# B&R Automation Studio project TD52 (part 140)

#### Ctr_OutVRDPCyclic.st
```iecst
(*******************************************************************************
Ctr_OutlVentRDP		controller engine room differential pressure with outlet ventilation fan(s)

This code is confidential and proprietary to the INNIO Company.
It may not be used in any form, or reproduced in any manner,
without the express written permission of the INNIO Company.
Copyright, INNIO Company, 2022

Customized modifications: -
------------------------

History:
-------
V4.04.0		06.10.2016	Stary			created
			02.11.2016	lettenb.		% scaling corr., cleanup
			15.11.2016  Stary		    added manual operation aux-control for outlet-ventilation
			04.01.2017  Stary           correction of task after test on simulator
V4.11.0		28.01.2022	Perktold		included plant controller upgrade

Specification       : PID-controller for outlet ventilation fan(s) to ensure a constant room differential pressure

Instructions for use: Modify release/X/external Y customized when needed
--------------------

Outstandings:
------------
(*******************************************************************************)

PROGRAM _CYCLIC

	(* Parameter *)
	Para.tCtr_OutlVE_RDP.W_set;
	Para.tCtr_OutlVE_RDP.W_set2;
	Para.tCtr_OutlVE_RDP.W_min;
	Para.tCtr_OutlVE_RDP.W_max;
	Para.tCtr_OutlVE_RDP.dW_up;
	Para.tCtr_OutlVE_RDP.dW_down;
	Para.tCtr_OutlVE_RDP.deadband;
	Para.tCtr_OutlVE_RDP.Y_min;
	Para.tCtr_OutlVE_RDP.Y_max;
	Para.tCtr_OutlVE_RDP.dY_max;
	Para.tCtr_OutlVE_RDP.Y_block;
	Para.tCtr_OutlVE_RDP.invert;
	Para.tCtr_OutlVE_RDP.Kp;
	Para.tCtr_OutlVE_RDP.Tn;
	Para.tCtr_OutlVE_RDP.Tv;
	Para.tCtr_OutlVE_RDP.Kp_GainScheduling;
	Para.tCtr_OutlVE_RDP.Tn_GainScheduling;
	Para.tCtr_OutlVE_RDP.Tv_GainScheduling;
	Para.tCtr_OutlVE_RDP.t_min_pulse_down;
	Para.tCtr_OutlVE_RDP.t_min_pulse_up;
	Para.tCtr_OutlVE_RDP.t_period_down;
	Para.tCtr_OutlVE_RDP.t_period_up;

	(* Time delay door-contact, to wait for correct measuring value room differential pressure after MSF --> avoid jump of Y *)
	TON_DC(IN := IN_VE.tER_DoorClosed.Di , PT := T#5s);
	bTON_DoorContact := TON_DC.Q;

	(* Input variables *)
	tCtr_OutlVE_RDP_In	 		:= VIS2MM.tCtr_OutlVE_RDP_In;

	(* Input from module *)
	tCtr_OutlVE_RDP_In.enable	:=	IN_VE.tPB2MM.bParaSetupOk		(* enable controller *)
							AND	    Para.bCtr_OutlVE_RDP
							AND     OUT_VE.tRel_ER_FC.Do
							AND	    RTM25
							AND     OUT_VE.tRel_ER_Fan.Do
							AND		bTON_DoorContact
							AND NOT MM2VIS.bMsg3367
							AND NOT MM2VIS.bMsg2705
							AND NOT bCtrER_YFix;

	tCtr_OutlVE_RDP_In.W_ext_Active		:= FALSE;		(* select external W *) //from visu
	tCtr_OutlVE_RDP_In.W_ext        	:= 0;
	tCtr_OutlVE_RDP_In.W_set2_Active	:= FALSE;		(*Input to define which internal setpoint will be used TRUE = use the 2nd set point | FALSE use the normal "1st" one*)
	tCtr_OutlVE_RDP_In.GainScheduling	:= 0.0;			(*Input for Gain Scheduling: 0.0 = use 100% of the Standard PID-Parameters | 1.0 = use 100% of the GainSched. PID Parameters | linear interpolation in between*)
	tCtr_OutlVE_RDP_In.Y_min_cust		:= -1.0;		(*"customized" Y-Min at the current moment (The existing Y-Min parameter is the global minimum. To have an effect Y_min_cust needs to be > the parameter | -1.0 = function not used*)
	tCtr_OutlVE_RDP_In.Y_max_cust		:= 1.0;			(*"customized" Y-Max at the current moment (The existing Y-Max parameter is the global maximum. To have an effect Y_max_cust needs to be < the parameter | 1.0 = function not used*)
	tCtr_OutlVE_RDP_In.Retrigger		:= FALSE;		(*a rising edge on this input signals the controller to retrigger - set W on X and force the Integrator to the current Y*)
	tCtr_OutlVE_RDP_In.A;								(*optional: feed forward Input*)

	(* Special operation-modes of PID-controller *)

		// Gas-pre-alarm/gas-alarm:
		    (* use of external Yset --> totally open the louver(s) *)
				IF IN_VE.bMsg1052 OR IN_VE.bMsg1053 THEN
					tCtr_OutlVE_RDP_In.Y_set_Active := TRUE;
					tCtr_OutlVE_RDP_In.Y_set := 1.0;
					RAMPE_Y_set_intern := FALSE;

		// Fire-alarm:
			(* use of external Yset --> totally close the louver(s) *)
				ELSIF IN_VE.bMsg1054 THEN
					tCtr_OutlVE_RDP_In.Y_set_Active := TRUE;
					tCtr_OutlVE_RDP_In.Y_set := 0.0;
					RAMPE_Y_set_intern := FALSE;

		// Engine room door-sensors tripped:
			(* use of internal Yset = last setpoint when ctr was active + slow PID-ramp *)
				ELSIF NOT bTON_DoorContact THEN
					tCtr_OutlVE_RDP_In.Y_set_Active := TRUE;
					Y_set_intern := rCtr_OutlVe_RDP_Y_old;  (* guilty for max. 15s, if doors are longer open then shutdown with bMsg3367 *)
					RAMPE_Y_set_intern := TRUE;

		// Measuring signal failure room differential pressure:
			(* use of internal Yset = ctr-signal from inlet ventilation + offset-para [13586] + slow PID-ramp *)
				ELSIF MM2VIS.bMsg2705 THEN
					tCtr_OutlVE_RDP_In.Y_set_Active := TRUE;
					Y_set_intern := tCtr_ER_Out.Y + (Para.rVent_SpeedDif);
					RAMPE_Y_set_intern := TRUE;

		// Manual operating auxiliaries control - Handbedienebene
				ELSIF (NOT tCtr_OutlVE_RDP_In.enable AND OUT_VE.tRel_ER_FC.Do AND IN_VE.tManAuxCtr.bER_OutlV_FC_Set) THEN
					tCtr_OutlVE_RDP_In.Y_set_Active  := TRUE;
					tCtr_OutlVE_RDP_In.Y_set         := IN_VE.tManAuxCtr.rER_OutlV_FC_Set;
					RAMPE_Y_set_intern := FALSE;

		// normal PID mode
				ELSE
					tCtr_OutlVE_RDP_In.Y_set_Active := FALSE;
					RAMPE_Y_set_intern := FALSE;
					Y_set_intern := tCtr_OutlVE_RDP_Out.Y;
				END_IF;

	(* slow PID-ramp *)
		RAMPE_R_0(enable := TRUE, In := Y_set_intern, Rise := 0.01, Sink := 0.01, TC_Time := 100);

		IF RAMPE_Y_set_intern THEN
			tCtr_OutlVE_RDP_In.Y_set := RAMPE_R_0.Out;
		END_IF

	tCtr_OutlVE_RDP_In.X := IN_VE.tPrDiff_ER.Ai;				(* select X *)

	(* add offset to Y *)
	xSigScal_R_CtrRDP_CtrER.X  := tCtr_ER_Out.Y;				(* scaling from setpoint ctr engine room to offset for use in outlet ventilation ctr *)
	xSigScal_R_CtrRDP_CtrER.X1 := Para.rScal_CtrInlVentER_Set_Min;
	xSigScal_R_CtrRDP_CtrER.X2 := Para.rScal_CtrInlVentER_Set_Max;
	xSigScal_R_CtrRDP_CtrER.Y1 := Para.rScal_OffSetMin_CtrOutlVent;
	xSigScal_R_CtrRDP_CtrER.Y2 := Para.rScal_OffSetMax_CtrOutlVent;
	xSigScal_R_CtrRDP_CtrER();

	xSigScal_R_CtrRDP_EngP.X  := IN_VE.rP_Act_Norm_Filt;		(* scaling from actual engine power to offset for use in outlet ventilation ctr *)
	xSigScal_R_CtrRDP_EngP.X1 := Para.rScal_PminEl;
	xSigScal_R_CtrRDP_EngP.X2 := Para.rScal_PmaxEl;
	xSigScal_R_CtrRDP_EngP.Y1 := Para.rScal_OffSetMin_Pel;
	xSigScal_R_CtrRDP_EngP.Y2 := Para.rScal_OffSetMax_Pel;
	xSigScal_R_CtrRDP_EngP();

	(* Input from Visualization via OPC *)
	tCtr_OutlVE_RDP_In.Y_man_Active;
	tCtr_OutlVE_RDP_In.Y_man;
	tCtr_OutlVE_RDP_In.X_min;
	tCtr_OutlVE_RDP_In.X_max;
	tCtr_OutlVE_RDP_In.Tune_quality;
	tCtr_OutlVE_RDP_In.Tune_PI;
	tCtr_OutlVE_RDP_In.Tune_PID;
	tCtr_OutlVE_RDP_In.Tune_start;
	tCtr_OutlVE_RDP_In.Tune_stop;
	tCtr_OutlVE_RDP_In.Tune_takeover;

	xCtr_OutlVE_RDP();

	(* Writing of actual Y on internal variable *)

	IF bTON_DoorContact THEN
		rCtr_OutlVe_RDP_Y_old	        := tCtr_OutlVE_RDP_Out.Y;	(* used as setpoint if engine room door-sensors have tripped *)
	END_IF;

	(* Output variables function block *)
	(* Output to module(s) *)

		// Control of outlet ventilation speed depending on ctr-signal inlet ventilation:
		// --> activation with parameter [13846]
			IF tCtr_OutlVE_RDP_In.enable AND Para.bCtr_RDP_OutlVE_Dep_InlVent AND NOT Para.bCtr_RDP_OutlVE_Dep_EngP THEN
				OUT_VE.tCtr_OutlVE_RDP_Set.Ao := LIMIT(0.0, tCtr_OutlVE_RDP_Out.Y + xSigScal_R_CtrRDP_CtrER.Y_SCAL, 1.0); (* analog out *)

		// Control of outlet ventilation speed depending on actual engine power:
		// --> activation with parameter [13847]
			ELSIF tCtr_OutlVE_RDP_In.enable AND Para.bCtr_RDP_OutlVE_Dep_EngP AND NOT Para.bCtr_RDP_OutlVE_Dep_InlVent THEN
				OUT_VE.tCtr_OutlVE_RDP_Set.Ao := LIMIT(0.0, tCtr_OutlVE_RDP_Out.Y + xSigScal_R_CtrRDP_EngP.Y_SCAL, 1.0); (* analog out *)

		// Control of outlet ventilation speed depending on inlet ventilation and actual engine power:
		// --> activation with parameter [1346+13847]
			ELSIF tCtr_OutlVE_RDP_In.enable AND Para.bCtr_RDP_OutlVE_Dep_InlVent AND Para.bCtr_RDP_OutlVE_Dep_EngP THEN
				OUT_VE.tCtr_OutlVE_RDP_Set.Ao := LIMIT(0.0, tCtr_OutlVE_RDP_Out.Y + xSigScal_R_CtrRDP_CtrER.Y_SCAL + xSigScal_R_CtrRDP_EngP.Y_SCAL, 1.0); (* analog out *)

			ELSE
				OUT_VE.tCtr_OutlVE_RDP_Set.Ao   := tCtr_OutlVE_RDP_Out.Y;		(* analog out *)
			END_IF;

	(* Output to Visualization via OPC *)
	MM2VIS.tCtr_OutlVE_RDP_Out		:= tCtr_OutlVE_RDP_Out;
	MM2VIS.rCtr_OutlVE_RDP_Set      := OUT_VE.tCtr_OutlVE_RDP_Set.Ao;
	VIS2MM.tCtr_OutlVE_RDP_In		:= tCtr_OutlVE_RDP_In;		(* write back to IN_struct for reset: Tune_takeover, X-display, ...!*)

	tCtr_OutlVE_RDP_Out.Active;
	tCtr_OutlVE_RDP_Out.Y;
	tCtr_OutlVE_RDP_Out.W;
	tCtr_OutlVE_RDP_Out.e;
	tCtr_OutlVE_RDP_Out.Kp_tune;
	tCtr_OutlVE_RDP_Out.Tn_tune;
	tCtr_OutlVE_RDP_Out.Tv_tune;
	tCtr_OutlVE_RDP_Out.status;
	tCtr_OutlVE_RDP_Out.Step_down;
	tCtr_OutlVE_RDP_Out.Step_up;

END_PROGRAM
```

#### Ctr_OutVRDPInit.st
```iecst
PROGRAM _INIT

	xCtr_OutlVE_RDP.pParameter 	:= ADR(Para.tCtr_OutlVE_RDP);
	xCtr_OutlVE_RDP.pInput 	 	:= ADR(tCtr_OutlVE_RDP_In);
	xCtr_OutlVE_RDP.pOutput	 	:= ADR(tCtr_OutlVE_RDP_Out);

	tCtr_OutlVE_RDP_In.AlwaysUseYRamp		:= TRUE;	(*If TRUE the Y signal will always limit the change rate via the according parameter | if FALSE the Y signal will jump in case the controller is disabled (blocked or set)*)
	tCtr_OutlVE_RDP_In.KeepYManAtBlock		:= TRUE;	(*If TRUE the controller will keep the Y-man value constant in case the controller is disabled (blocked or set) | If FALSE the blocked or set value will override the Y-man value*)
	tCtr_OutlVE_RDP_In.Y_min_cust			:= -1.0;	(*"customized" Y-Min at the current moment (The existing Y-Min parameter is the global minimum. To have an effect Y_min_cust needs to be > the parameter | -1.0 = function not used*)
	tCtr_OutlVE_RDP_In.Y_max_cust			:=  1.0;	(*"customized" Y-Max at the current moment (The existing Y-Max parameter is the global maximum. To have an effect Y_max_cust needs to be < the parameter | 1.0 = function not used*)
	tCtr_OutlVE_RDP_In.StepperMode			:= FALSE;	(* TRUE = use PWM-Mode (standard mode until 4.10) | FALSE = use continuous servo drive *)

END_PROGRAM
```

#### Ctr_OutVRDP.var
```iecst
VAR
	rCtr_OutlVe_RDP_Y_old : REAL; (*write the actual Y on this internal variable*)
	xSigScal_R_CtrRDP_EngP : xSigScal_R := (0);
	xSigScal_R_CtrRDP_CtrER : xSigScal_R := (0);
	TON_DC : TON; (*TON door contact*)
	RAMPE_R_0 : RAMPE_R := (0);
	RAMPE_Y_set_intern : BOOL := 0;
	Y_set_intern : REAL;
END_VAR
```

### Program Logical/Ventilation/Ctr_ER (IEC, version 4.11.0) - controller engine room temperature

#### Ctr_ERCyclic.st
```iecst
(*******************************************************************************
Ctr_ER		controller engine room temperature

This code is confidential and proprietary to the INNIO Company.
It may not be used in any form, or reproduced in any manner,
without the express written permission of the INNIO Company.
Copyright, INNIO Company, 2022

Customized modifications: -
------------------------

History:
-------
V0.00.0		17.04.2012	lettenbichler	created
			23.11.2012	lettenbichler	write back to IN_struct added (zengerer)
V3.99.0		24.06.2013	lettenbichler	tCtr_ER_In.Y_set := 100.0 -> 1.0, bugfix
V4.00.0		22.05.2015					tCtr_ER_In.X: Para.bT_InAirER_Active added(room vent.to 100% if no sensor active)
V4.03.0 	07.08.2015  Denk			Manual operating auxiliaries control functionality added
V4.05.0 	20.09.2017	Messner			Active Cooling Program added
V4.11.0		28.01.2022	Perktold		included plant controller upgrade

Instructions for use:
--------------------

Outstandings:
------------
(*******************************************************************************)

PROGRAM _CYCLIC

	(* Parameter *)
	Para.tCtr_ER.W_set;
	Para.tCtr_ER.W_set2;
	Para.tCtr_ER.W_min;
	Para.tCtr_ER.W_max;
	Para.tCtr_ER.dW_up;
	Para.tCtr_ER.dW_down;
	Para.tCtr_ER.deadband;
	Para.tCtr_ER.Y_min;
	Para.tCtr_ER.Y_max;
	Para.tCtr_ER.dY_max;
	Para.tCtr_ER.Y_block;
	Para.tCtr_ER.invert;
	Para.tCtr_ER.Kp;
	Para.tCtr_ER.Tn;
	Para.tCtr_ER.Tv;
	Para.tCtr_ER.Kp_GainScheduling;
	Para.tCtr_ER.Tn_GainScheduling;
	Para.tCtr_ER.Tv_GainScheduling;
	Para.tCtr_ER.t_min_pulse_down;
	Para.tCtr_ER.t_min_pulse_up;
	Para.tCtr_ER.t_period_down;
	Para.tCtr_ER.t_period_up;

	(* Input variables *)
	tCtr_ER_In	 				:= VIS2MM.tCtr_ER_In;

	(* Input from module *)
	tCtr_ER_In.enable			:=	IN_VE.tPB2MM.bParaSetupOk		(* enable controller *)
							AND		Para.bCtr_ER
							AND 	OUT_VE.tRel_ER_FC.Do
							AND	  ((RTM25 AND OUT_VE.tRel_ER_Fan.Do) OR (Para.bER_VentColdCountryMode AND NOT OUT_VE.tSet_ER_Fan_Min.Do))
							AND NOT MS_LUE
							AND NOT bCtrER_YFix;

	tCtr_ER_In.W_ext_Active	:= tCtr_ER_In.W_ext_Active OR TRUE;		(* select external W *) //from visu

	IF IN_VE.bEng_Aux_Dem_CDR THEN
		tCtr_ER_In.W_ext :=	 Para.rT_CtrER_WexRun;					(* external W *)
	ELSIF IN_VE.bACP_AirER_Dem THEN
		tCtr_ER_In.W_ext :=	 Para.rT_ACP_AirER_sp;					(* ACP  Room Temperature set point *)
	ELSE
		tCtr_ER_In.W_ext :=	 Para.rT_CtrER_WexStop;
	END_IF;
	tCtr_ER_In.W_set2_Active	:= FALSE;		(*Input to define which internal setpoint will be used TRUE = use the 2nd set point | FALSE use the normal "1st" one*)
	tCtr_ER_In.GainScheduling	:= 0.0;			(*Input for Gain Scheduling: 0.0 = use 100% of the Standard PID-Parameters | 1.0 = use 100% of the GainSched. PID Parameters | linear interpolation in between*)
	tCtr_ER_In.Y_min_cust		:= -1.0;		(*"customized" Y-Min at the current moment (The existing Y-Min parameter is the global minimum. To have an effect Y_min_cust needs to be > the parameter | -1.0 = function not used*)
	tCtr_ER_In.Y_max_cust		:= 1.0;			(*"customized" Y-Max at the current moment (The existing Y-Max parameter is the global maximum. To have an effect Y_max_cust needs to be < the parameter | 1.0 = function not used*)
	tCtr_ER_In.Retrigger		:= FALSE;		(*a rising edge on this input signals the controller to retrigger - set W on X and force the Integrator to the current Y*)
	tCtr_ER_In.A;								(*optional: feed forward Input*)

	IF bCtrER_YFix = TRUE THEN
		tCtr_ER_In.Y_set_Active	:= bCtrER_YFix; 	 				(* select external Y *)
		tCtr_ER_In.Y_set		:= 1.0;
	ELSIF (	NOT tCtr_ER_In.enable 									(* Manual operating auxiliaries control - Handbedienebene *)
			AND OUT_VE.tRel_ER_FC.Do
			AND IN_VE.tManAuxCtr.bER_FC_Set) THEN
		tCtr_ER_In.Y_set_Active := TRUE;
		tCtr_ER_In.Y_set		:= IN_VE.tManAuxCtr.rER_FC_Set;
	ELSE
		tCtr_ER_In.Y_set_Active	:= FALSE;
	END_IF;

	IF Para.bER_VentColdCountryMode AND IN_VE.bEng_Aux_Dem_CDR (*AND Para.bT_InAirER_Active*) THEN
		tCtr_ER_In.X :=	MAX(rT_AirER, IN_VE.rT_Ch_T1LP_Avg);		(* select X *)
	ELSE
		tCtr_ER_In.X :=	    rT_AirER;
	END_IF;
	tCtr_ER_In.A := 0;

	(* Input from Visualization via OPC *)
	tCtr_ER_In.Y_man_Active;
	tCtr_ER_In.Y_man;
	tCtr_ER_In.X_min;
	tCtr_ER_In.X_max;
	tCtr_ER_In.Tune_quality;
	tCtr_ER_In.Tune_PI;
	tCtr_ER_In.Tune_PID;
	tCtr_ER_In.Tune_start;
	tCtr_ER_In.Tune_stop;
	tCtr_ER_In.Tune_takeover;

	xCtr_ER();

	(* Output variables function block *)
	(* Output to module(s) *)
	OUT_VE.tER_FC_Set.Ao 	:= tCtr_ER_Out.Y;	(* analog out *)

	(* Output to Visualization via OPC *)
	MM2VIS.tCtr_ER_Out		:= tCtr_ER_Out;
	VIS2MM.tCtr_ER_In		:= tCtr_ER_In;		(* write back to IN_struct for reset: Tune_takeover, X-display, ...!*)

	tCtr_ER_Out.Active;
	tCtr_ER_Out.Y;
	tCtr_ER_Out.W;
	tCtr_ER_Out.e;
	tCtr_ER_Out.Kp_tune;
	tCtr_ER_Out.Tn_tune;
	tCtr_ER_Out.Tv_tune;
	tCtr_ER_Out.status;
	tCtr_ER_Out.Step_down;
	tCtr_ER_Out.Step_up;

END_PROGRAM
```

#### Ctr_ERInit.st
```iecst
PROGRAM _INIT

	xCtr_ER.pParameter 	:= ADR(Para.tCtr_ER);
	xCtr_ER.pInput 	 	:= ADR(tCtr_ER_In);
	xCtr_ER.pOutput	 	:= ADR(tCtr_ER_Out);

	tCtr_ER_In.AlwaysUseYRamp		:= TRUE;	(*If TRUE the Y signal will always limit the change rate via the according parameter | if FALSE the Y signal will jump in case the controller is disabled (blocked or set)*)
	tCtr_ER_In.KeepYManAtBlock		:= TRUE;	(*If TRUE the controller will keep the Y-man value constant in case the controller is disabled (blocked or set) | If FALSE the blocked or set value will override the Y-man value*)
	tCtr_ER_In.Y_min_cust			:= -1.0;	(*"customized" Y-Min at the current moment (The existing Y-Min parameter is the global minimum. To have an effect Y_min_cust needs to be > the parameter | -1.0 = function not used*)
	tCtr_ER_In.Y_max_cust			:=  1.0;	(*"customized" Y-Max at the current moment (The existing Y-Max parameter is the global maximum. To have an effect Y_max_cust needs to be < the parameter | 1.0 = function not used*)
	tCtr_ER_In.StepperMode			:= FALSE;	(* TRUE = use PWM-Mode (standard mode until 4.10) | FALSE = use continuous servo drive *)

END_PROGRAM
```

### Program Logical/Ventilation/vis_VE (IEC, version 4.05.1) - visualization

#### vis_VECyclic.st
```iecst
(*******************************************************************************
vis			visualization

This code is confidential and proprietary to the INNIO Company.
It may not be used in any form, or reproduced in any manner,
without the express written permission of the INNIO Company.
Copyright, INNIO Company, 2019

Customized modifications: -
------------------------

History:
-------
V3.99.0	24.04.2012	lettenb.	new
V4.00.0	02.06.2014				MM2VIS.bRel_ER_Fan: OUT_VE.tRel_ER_Fan.Do -> OUT_VE.tRel_ER_FC.Do, bugfix
V4.03.0 19.11.2015  Stary       added MM2VIS.rPrDiff_ER :=  IN_VE.tPrDiff_ER.Ai;
V4.04.0 21.10.2016  Stary       added MM2VIS.bCtrER_YFix :=  bCtrER_YFix; for visualization of BOP on HMI
V4.04.0 22.10.2016  Stary       added status-messages of fire-protection flaps
		07.11.2016	lettenb.	MM2VIS.rP_Red_T_InAirER_Norm removed(see:OpState)
V4.04.0 09.01.2017  Stary       correction of line 43 (was written on status of fire prot flap outlet air 1 too)
V4.05.1 01.03.2018	lettenb.	Pos_InlLou1_OK, Pos_InlLou2_OK, Pos_OutlLou1_OK added(kluckner), bugfix

Instructions for use:
--------------------
Outstandings:
------------
*******************************************************************************)
PROGRAM _CYCLIC

	MM2VIS.rT_AirER							:=	rT_AirER;
	MM2VIS.rPrDiff_ER           			:=  IN_VE.tPrDiff_ER.Ai;

	MM2VIS.bInAirER_Lou1Opened				:=	IN_VE.tInAirER_Lou1Opened.Di OR Pos_InlLou1_OK;
	MM2VIS.bInAirER_Lou2Opened				:=	IN_VE.tInAirER_Lou2Opened.Di OR Pos_InlLou2_OK;
	MM2VIS.bOutAirER_LouOpened				:=	IN_VE.tOutAirER_LouOpened.Di OR Pos_OutlLou1_OK OR Pos_OutlLou2_OK;
	MM2VIS.bInAirER_Fan1DemOn				:=	OUT_VE.tInAirER_Fan1DemOn.Do;
	MM2VIS.bInAirER_Fan2DemOn				:=	OUT_VE.tInAirER_Fan2DemOn.Do;
	MM2VIS.bInAirER_FanSet100				:=	IN_VE.bInAirER_FanSet100;
	MM2VIS.bRel_ER_Fan						:=	OUT_VE.tRel_ER_FC.Do;
	MM2VIS.bCtrER_YFix						:=  bCtrER_YFix;
	MM2VIS.bFireProtFlap1_InlAir_Opened 	:=  IN_VE.tFireProtFlap1_InlAir_Opened.Di AND NOT IN_VE.tFireProtFlap1_InlAir_Closed.Di;
	MM2VIS.bFireProtFlap2_InlAir_Opened 	:=  IN_VE.tFireProtFlap2_InlAir_Opened.Di AND NOT IN_VE.tFireProtFlap2_InlAir_Closed.Di;
	MM2VIS.bFireProtFlap1_OutlAir_Opened 	:=  IN_VE.tFireProtFlap1_OutlAir_Opened.Di AND NOT IN_VE.tFireProtFlap1_OutlAir_Closed.Di;
	MM2VIS.bFireProtFlap2_OutlAir_Opened 	:=  IN_VE.tFireProtFlap2_OutlAir_Opened.Di AND NOT IN_VE.tFireProtFlap2_OutlAir_Closed.Di;

END_PROGRAM
```

### Program Logical/Ventilation/MsgVE (IEC, version 4.13.0) - messages

#### MsgVECyclic.st
```iecst
(*******************************************************************************
MsgVE	 			ventilation messages

This code is confidential and proprietary to the INNIO Company.
It may not be used in any form, or reproduced in any manner,
without written permission of the INNIO Company.
Copyright, INNIO Company, 2022

Customized modifications: -
------------------------

History:
-------
V0.01.0	02.11.2011	lettenb.	new
		18.09.2012	lettenb.	rT_AirER_Customized added (request zengerer)
V3.40.0	17.12.2012	lettenb.	1138 DI_ERV_Op added, preparation for air flow sensor, ATEX
								3224 .PTON := T#0s -> 2s; (W3223 MS & W3224 comes at the same time) bugfix
V3.99.0	19.02.2013	lettenb.	update
		24.05.2013				reset OUT_xx.txx2AB.bGnlTripx changed
V4.00.0	31.01.2014				3367 added, eng.room vent.monit.V3.50
V4.00.1	14.05.2014	lettenb.	1138 var 3/4: FG_FU, ZLVST1 added (MRL kalte laender)
		12.06.2014				3224 xTON_GCB_On.PT:= T#30s -> 300s, bugfix
V4.00.2	16.02.2015				3152,3223 enable with IN_VE.tPB2MM.bSys_Run
V4.03.0 03.08.2015  Stary       added new alarms 2701-2709 FOR controlled louvers
					lettenb.	xMsg2704.Enable: Para.bInlVent_Ctr_OutlLou_Active -> Para.bOutlVent_Ctr_OutlLou_Active, bugfix
		30.09.2015  Stary       2120 tAuxV_Aux_ok added
		23.12.2015	lettenb.	1138 M_DREHZ -> (IN_VE.bEng_Dem OR IN_VE.tEng_Run.Do) to avoid msg after mains failure(restart ability)
V4.04.0 07.07.2016	lettenb.	2630 added(substitution for 1176 in wrong module(CH) tDPr_InAirFilt_Hi -> tDPr_InAirFiltERV_Hi), bugfix
V4.04.0 27.09.2016  Stary       splitted up existing summarized alarms 1138+2120 for ventilation and added single alarms for inlet/outlet --> new messages 2295,2296,2795-2798
		02.11.2016	Tinello		3223 und 3224 deleted --> moved to modul CH
V4.04.0 25.01.2017  Stary   	bugfix after pilot-engines:
								Enable of bMsg2701-bMsg2704 --> deleted Para.bInlVent_Ctr_InlLou_Active cause measuring singnal failure now indepedend OF ventilation type
		01.02.2017	lettenb.	xTON_MonAuxV double function call removed
V4.05.0 30.06.2017	lettenb.	bAuxRel_Louvers added acc. faststart option
		21.12.2017	lettenb.	1138, 2295, 2296 enable alarms depending on existing Di's (stary), bugfix
		22.12.2017	lettenb.	comment added: Safety-related application software source code (EN 13849-1 / 4.6.3)
		22.01.2018	lettenb.	1138 Pos_InlLou1_OK, Pos_InlLou2_OK, Pos_OutlLou1_OK, Pos_OutlLou2_OK added, bugfix
		22.01.2018	lettenb.	3152 bParaSetupOk added TO avoid message at plc startup
		30.01.2018	lettenb.	2706,2707 time delay 10s(fahringer/stary)
V4.06.0	16.07.2018	Perktold,	2968 and 2969 Air inlet/outlet louver status signal failure added
V4.07.0 25.02.2019	Stary/lett. 1138,2295,2296 bAuxRel_FireProtFlaps: FireProtFlap feedback signals included in aux.release, safety case
								2295,2296 bAuxRel_Louvers_... added(same as 1138), xTON_MonAuxV double function call removed, bugfix
V4.10.0 25.01.2021	lettenb.	engine room ventilation not ready - block engine start as long as failure is active, added from task Vent_ER (request fahringer), bugfix
								2120,2795,2796 safety code remark added (request fahringer)
V4.12.0 07.12.2022	lettenb.	2706: IN_VE.tEng_Run.Do added, aggreko -> jenb.standard, #954
V4.13.0 18.03.2024	Bacci		2295: trip used when inlet louvers demanded but not responding (90s)
V4.14.0 10.12.2024	Nagy		New warning 2472 High Temperature Warning and Alarm 9401 Louvers 2024-226

Instructions for use:
--------------------
1) declare alarm with function block "Alm"
	declare buffert alarm bit bMsg<message number>

2) use template to create a new alarm,
   substitue 0000 by alarm number and make settings:

	xMsg0000.Enable		:=	TRUE;		enable/disable alarm
	xMsg0000.Set		:=	FALSE;		alarm set condition
	xMsg0000.PT			:=	T#0s;		alarm delay time
	xMsg0000.Prio		:=	1;			alarm priority: 1-3 = trip, 4 = warning
	xMsg0000.RiskClass	:=	3;			risk class for remote alarm reset acc.TI 1100-0111
	xMsg0000.Reset		:=	FALSE;		FALSE: for all standard alarms	prio 1,2,3 and warnings prio 4
										TRUE : for autoreset alarms

	bMsg0000			:=	xMsg0000.Q;	connect buffert alarm bit for VIS and control

3)  expand INIT

Outstandings:
------------
change bGnlTrip_VE --> bGnlTrip
(*******************************************************************************)
PROGRAM _CYCLIC

	(* reset general trip *)
	OUT_VE.tVE2AB.bGnlTrip1		:=	FALSE;
	OUT_VE.tVE2AB.bGnlTrip2		:=	FALSE;
	OUT_VE.tVE2AB.bGnlTrip3		:=	FALSE;
	OUT_VE.tVE2AB.bGnlWarning	:=	FALSE;
	OUT_VE.tVE2AB.bTriptype1	:=	FALSE;
	OUT_VE.tVE2AB.bTriptype2	:=	FALSE;
	OUT_VE.tVE2AB.bTriptype3	:=	FALSE;

	(*  1135 engine room temperature high *)
	xTON_RoomTemp.IN :=   ((NOT MM2VIS.bMsg3152) AND bT_AirER_Hi)
						OR (NOT Para.bVISA  AND NOT IN_VE.tT_AirER_Ext_Hi.Di);
	xTON_RoomTemp.PT :=  T#30s;
	xTON_RoomTemp();
	T_RTM := xTON_RoomTemp.Q;

	xMsg1135.Enable		:=	TRUE;
	xMsg1135.Set		:= (T_RTM      AND(NOT IN_VE.bEng_Dem_EPS OR IN_VE.bOnly_Island))
						OR (Para.bVISA AND NOT IN_VE.tT_AirER_Ext_Hi.Di);
	xMsg1135.PT			:=	T#0s;

	RTM_VISA := NOT IN_VE.tT_AirER_Ext_Hi.Di  OR (RTM_VISA AND xMsg1135.Q);
	IF Para.bVISA AND RTM_VISA THEN
		xMsg1135.Prio	:=	2;
	ELSE
		xMsg1135.Prio	:=	3;
	END_IF;
	xMsg1135.RiskClass	:=	0;		(* TI 1100-0111 *)
	xMsg1135.Reset		:=	FALSE;
	xMsg1135();
	MM2VIS.bMsg1135	    :=	xMsg1135.Q;

	(*  2472 engine room temperature high warning*)
	xMsg2472.Enable		:=	TRUE;
	xMsg2472.Set		:= bT_AirER_Hi_Wr AND (NOT IN_VE.bEng_Dem_EPS OR IN_VE.bOnly_Island)
	OR (Para.bVISA AND NOT IN_VE.tT_AirER_Ext_Hi.Di);
	xMsg2472.PT			:=	T#1s;
	xMsg2472.Prio		:=	4;
	xMsg2472.RiskClass	:=	0;		(* TI 1100-0111 *)
	xMsg2472.Reset		:=	FALSE;
	xMsg2472();
	MM2VIS.bMsg2472	    :=	xMsg2472.Q;

	(********************************************************************************************************************
	Safety-related application software source code (EN 13849-1 / 4.6.3): BEGIN
	*********************************************************************************************************************)
	(*  1138 engine room fan failure trip (W2120) *)
	bERV_AirFlowMon_Off :=	(IN_VE.tInAirER_Lou1Opened.Di OR IN_VE.tInAirER_Lou2Opened.Di OR IN_VE.tOutAirER_LouOpened.Di OR Pos_InlLou1_OK OR Pos_InlLou2_OK OR Pos_OutlLou1_OK OR Pos_OutlLou2_OK)
					 AND NOT(IN_VE.bEng_Dem OR IN_VE.tEng_Run.Do); 		(* monit.off for reason of natural air flow with open louvers *)
	xTON_StartERV(IN:= IN_VE.bEng_Aux_Dem_CDR, PT:= T#30s);				(* startverzoegerung fuer ueberwachung *)

	IF    Para.bERV_AirFlowMon_Active AND Para.bInAirER_Fan_FU THEN
			(* var: flow sensor, stationaeranlage, container BR6	*)
			(* var: stationaeranlage, steuerung RL durch GEJ inkl. Rueckmeldung RL in Betrieb (flow switch od.IFL 56.32) *)
		xTON_ERV_On(IN:=      FG_FU                        AND NOT IN_VE.tERV_Op.Di AND NOT bERV_AirFlowMon_Off, PT:= T#15s);(* delay on:  eng.room vent.ok/air flow monitoring *)
		xTON_ERV_Of(IN:=  NOT FG_FU                        AND     IN_VE.tERV_Op.Di AND NOT bERV_AirFlowMon_Off, PT:= T#5m); (* delay off: change contact check *)
	ELSIF Para.bERV_AirFlowMon_Active AND NOT Para.bInAirER_Fan_FU THEN
		xTON_ERV_On(IN:=      OUT_VE.tInAirER_Fan1DemOn.Do AND NOT IN_VE.tERV_Op.Di AND NOT bERV_AirFlowMon_Off, PT:= T#15s);(* delay on:  eng.room vent.ok/air flow monitoring *)
		xTON_ERV_Of(IN:=  NOT OUT_VE.tInAirER_Fan1DemOn.Do AND     IN_VE.tERV_Op.Di AND NOT bERV_AirFlowMon_Off, PT:= T#5m); (* delay off: change contact check *)
	ELSIF Para.bInAirER_Fan_FU THEN
			(* var: FU=RUN, ohne luftstromwaechter *)
		xTON_ERV_On(IN:=      FG_FU   					   AND NOT IN_VE.tERV_Op.Di AND    (IN_VE.bEng_Dem OR IN_VE.tEng_Run.Do), PT:= T#15s);
		xTON_ERV_Of(IN:= FALSE, PT:= T#5m);
	ELSE	(* var: lueftung in betrieb, ohne FU, ohne luftstromwaechter *)
		xTON_ERV_On(IN:=      OUT_VE.tInAirER_Fan1DemOn.Do AND NOT IN_VE.tERV_Op.Di AND    (IN_VE.bEng_Dem OR IN_VE.tEng_Run.Do), PT:= T#15s);
		xTON_ERV_Of(IN:= FALSE, PT:= T#5m);
	END_IF;
			(* keine ERV: 	para bERV_AirFlowMon_Active (default =0) => OFF
							para bAirInVentF (default=1) n.r.,
							DI_ERV_Op (default = 1) nicht belegt *)

	bAuxRel_Louvers := (IN_VE.tOutAirER_LouOpened.Di AND IN_VE.tInAirER_Lou1Opened.Di)
					OR((Pos_InlLou1_OK OR Pos_InlLou2_OK) AND (Pos_OutlLou1_OK OR Pos_OutlLou2_OK));

	bAuxRel_FireProtFlaps := IN_VE.tFireProtFlap1_InlAir_Opened.Di  AND IN_VE.tFireProtFlap2_InlAir_Opened.Di AND
							 IN_VE.tFireProtFlap1_OutlAir_Opened.Di AND IN_VE.tFireProtFlap2_OutlAir_Opened.Di;

	xTOF_EngDemEPS(IN:= IN_VE.bEng_Dem_EPS AND NOT IN_VE.tGCB_On.Di, PT:= T#60s);
	bNoMon4BlackStart := xTOF_EngDemEPS.Q AND IN_VE.bEng_Dem_EPS; //T14

	xMsg1138.Enable		:=	IN_VE.tERV_Op.GoodQual;
	xMsg1138.Set		:= (NOT bNoMon4BlackStart AND  ((xTON_ERV_On.Q AND xTON_StartERV.Q)
                                                     OR  xTON_ERV_Of.Q))
						OR (IN_VE.bFS_Act AND xTON_StartERV.Q AND NOT bAuxRel_Louvers)
						OR (IN_VE.bFS_Act AND xTON_StartERV.Q AND NOT bAuxRel_FireProtFlaps);
	xMsg1138.PT			:=	T#0s;
	xMsg1138.Prio		:=	3;
	xMsg1138.RiskClass	:=	4;
	xMsg1138.Reset		:=	FALSE;
	xMsg1138();
	MM2VIS.bMsg1138 	:=	xMsg1138.Q;
	(********************************************************************************************************************
	Safety-related application software source code (EN 13849-1 / 4.6.3): END
	*********************************************************************************************************************)

	(********************************************************************************************************************
	Safety-related application software source code (EN 13849-1 / 4.6.3): BEGIN
	*********************************************************************************************************************)
	(*  2120 engine room fan failure *)
	xTON_MonAuxV(IN:= IN_VE.tGCB_On.Di, PT:= T#60s);		(* release monitoring engine room fan failure *)

	IF Para.bInAirER_Fan_FU THEN
		xTON_ERV.IN			:= (NOT IN_VE.tER_Ext_Err.Di AND     IN_VE.tAuxV_Supply_Ok.Di AND IN_VE.tAuxV_Aux_ok.Di)
							OR (    xTON_MonAuxV.Q	     AND(NOT IN_VE.tAuxV_Supply_Ok.Di
														  OR NOT IN_VE.tAuxV_Aux_ok.Di));
	ELSE
		xTON_ERV.IN			:=  NOT IN_VE.tER_Ext_Err.Di;
	END_IF;
	xTON_ERV(PT:= T#12s);

	xMsg2120.Enable		:=	TRUE;
	xMsg2120.Set		:=	xTON_ERV.Q;
	xMsg2120.PT			:=	T#0s;
	xMsg2120.Prio		:=	4;
	xMsg2120.RiskClass	:=	4;
	xMsg2120.Reset		:=	FALSE;
	xMsg2120();
	MM2VIS.bMsg2120     :=	xMsg2120.Q;

	(* engine room ventilation not ready - block engine start as long as failure is active *)
	OUT_VE.bERV_NotRdy := xMsg2120.Set OR xMsg2795.Set OR xMsg2796.Set;
	(********************************************************************************************************************
	Safety-related application software source code (EN 13849-1 / 4.6.3): END
	*********************************************************************************************************************)

	(********************************************************************************************************************
	Safety-related application software source code (EN 13849-1 / 4.6.3): BEGIN
	*********************************************************************************************************************)
	(*  2295 engine room ventilation failure inlet air *)
	bERV_InlAirFlowMon_Off := (IN_VE.tInAirER_Lou1Opened.Di OR IN_VE.tInAirER_Lou2Opened.Di OR Pos_InlLou1_OK OR Pos_InlLou2_OK)
					  AND NOT (IN_VE.bEng_Dem OR IN_VE.tEng_Run.Do); 	(* monit.off for reason of natural air flow with open louvers *)
	xTON_StartERV(IN:= IN_VE.bEng_Aux_Dem_CDR, PT:= T#30s);				(* startverzoegerung fuer ueberwachung *)

	IF    Para.bERV_AirFlowMon_Active AND Para.bInAirER_Fan_FU THEN
		(* var: flow sensor, stationaeranlage, container BR6	*)
		(* var: stationaeranlage, steuerung RL durch GEJ inkl. Rueckmeldung RL in Betrieb *)
		xTON_ERV_Inl_On(IN:=      FG_FU                        AND NOT IN_VE.tERV_InlAir_Op.Di AND NOT bERV_InlAirFlowMon_Off, PT:= T#15s);(* delay on:  eng.room inl.vent.ok/air flow monitoring *)
		xTON_ERV_Inl_Of(IN:=  NOT FG_FU                        AND     IN_VE.tERV_InlAir_Op.Di AND NOT bERV_InlAirFlowMon_Off, PT:= T#5m); (* delay off: change contact check *)
	ELSIF Para.bERV_AirFlowMon_Active AND NOT Para.bInAirER_Fan_FU THEN
		xTON_ERV_Inl_On(IN:=      OUT_VE.tInAirER_Fan1DemOn.Do AND NOT IN_VE.tERV_InlAir_Op.Di AND NOT bERV_InlAirFlowMon_Off, PT:= T#15s);(* delay on:  eng.room inl.vent.ok/air flow monitoring *)
		xTON_ERV_Inl_Of(IN:=  NOT OUT_VE.tInAirER_Fan1DemOn.Do AND     IN_VE.tERV_InlAir_Op.Di AND NOT bERV_InlAirFlowMon_Off, PT:= T#5m); (* delay off: change contact check *)
	ELSIF Para.bInAirER_Fan_FU THEN
		(* var: FU=RUN, ohne luftstromwaechter *)
		xTON_ERV_Inl_On(IN:=      FG_FU   					   AND NOT IN_VE.tERV_InlAir_Op.Di AND    (IN_VE.bEng_Dem OR IN_VE.tEng_Run.Do), PT:= T#15s);
		xTON_ERV_Inl_Of(IN:= FALSE, PT:= T#5m);
	ELSE	(* var: lueftung in betrieb, ohne FU, ohne luftstromwaechter *)
		xTON_ERV_Inl_On(IN:=      OUT_VE.tInAirER_Fan1DemOn.Do AND NOT IN_VE.tERV_InlAir_Op.Di AND    (IN_VE.bEng_Dem OR IN_VE.tEng_Run.Do), PT:= T#15s);
		xTON_ERV_Inl_Of(IN:= FALSE, PT:= T#5m);
	END_IF;

	bAuxRel_Louvers_InlAir       := IN_VE.tInAirER_Lou1Opened.Di OR Pos_InlLou1_OK OR Pos_InlLou2_OK;
	bAuxRel_FireProtFlaps_InlAir := IN_VE.tFireProtFlap1_InlAir_Opened.Di AND IN_VE.tFireProtFlap2_InlAir_Opened.Di;

	xTOF_EngDemEPS(IN:= IN_VE.bEng_Dem_EPS AND NOT IN_VE.tGCB_On.Di, PT:= T#60s);
	bNoMon4BlackStart := xTOF_EngDemEPS.Q AND IN_VE.bEng_Dem_EPS; //T14

	xTON_InAirER_LouFail(IN:= (OUT_VE.tInAirER_Lou1DemOpen.Do OR OUT_VE.tInAirER_Lou2DemOpen.Do OR OUT_VE.tCtr_InlLou_Set.Ao > 0.5) AND NOT OUT_VE.bInLouRelVE AND xOpMode.Stop,  PT:= T#90s);		(* Inlet louver required and not opened *)

	xMsg2295.Enable		:=	IN_VE.tERV_InlAir_Op.GoodQual OR (xOpMode.Stop AND (xTON_InAirER_LouFail.Q OR MM2VIS.bMsg2295));
	xMsg2295.Set		:=	(NOT bNoMon4BlackStart AND ((xTON_ERV_Inl_On.Q AND xTON_StartERV.Q)
						    OR  xTON_ERV_Inl_Of.Q))
					        OR (IN_VE.bFS_Act AND xTON_StartERV.Q AND NOT bAuxRel_Louvers_InlAir)
	                        OR (IN_VE.bFS_Act AND xTON_StartERV.Q AND NOT bAuxRel_FireProtFlaps_InlAir)
							OR xTON_InAirER_LouFail.Q;
	xMsg2295.PT			:=	T#0s;
	xMsg2295.Prio		:=	3;
	xMsg2295.RiskClass	:=	10;
	xMsg2295.Reset		:=	FALSE;
	xMsg2295();
	MM2VIS.bMsg2295	    :=	xMsg2295.Q;
	OUT_VE.bMsg2295	    :=	xMsg2295.Q;

	(*  2296 engine room ventilation failure outlet air *)
	bERV_OutlAirFlowMon_Off := (IN_VE.tOutAirER_LouOpened.Di OR Pos_OutlLou1_OK OR Pos_OutlLou2_OK)
					   AND NOT (IN_VE.bEng_Dem OR IN_VE.tEng_Run.Do); (* monit.off for reason of natural air flow with open louvers *)
	xTON_StartERV(IN:= IN_VE.bEng_Aux_Dem_CDR, PT:= T#30s);				(* startverzoegerung fuer ueberwachung *)

	IF    Para.bERV_AirFlowMon_Active AND Para.bOutAirER_Fan_FU THEN
		(* var: flow sensor, stationaeranlage, container BR6	*)
		(* var: stationaeranlage, steuerung RL durch GEJ inkl. Rueckmeldung RL in Betrieb *)
		xTON_ERV_Outl_On(IN:=      FG_FU                          AND NOT IN_VE.tERV_OutlAir_Op.Di AND NOT bERV_OutlAirFlowMon_Off, PT:= T#15s);(* delay on:  eng.room outl.vent.ok/air flow monitoring *)
		xTON_ERV_Outl_Of(IN:=  NOT FG_FU                          AND     IN_VE.tERV_OutlAir_Op.Di AND NOT bERV_OutlAirFlowMon_Off, PT:= T#5m); (* delay off: change contact check *)
	ELSIF Para.bERV_AirFlowMon_Active AND NOT Para.bOutAirER_Fan_FU THEN
		xTON_ERV_Outl_On(IN:=      OUT_VE.tOutAirER_LouDemOpen.Do AND NOT IN_VE.tERV_OutlAir_Op.Di AND NOT bERV_OutlAirFlowMon_Off, PT:= T#15s);(* delay on:  eng.room outl.vent.ok/air flow monitoring *)
		xTON_ERV_Outl_Of(IN:=  NOT OUT_VE.tOutAirER_LouDemOpen.Do AND     IN_VE.tERV_OutlAir_Op.Di AND NOT bERV_OutlAirFlowMon_Off, PT:= T#5m); (* delay off: change contact check *)
	ELSIF Para.bOutAirER_Fan_FU THEN
		(* var: FU=RUN, ohne luftstromwaechter *)
		xTON_ERV_Outl_On(IN:=      FG_FU   					      AND NOT IN_VE.tERV_OutlAir_Op.Di AND    (IN_VE.bEng_Dem OR IN_VE.tEng_Run.Do), PT:= T#15s);
		xTON_ERV_Outl_Of(IN:= FALSE, PT:= T#5m);
	ELSE	(* var: lueftung in betrieb, ohne FU, ohne luftstromwaechter *)
		xTON_ERV_Outl_On(IN:=      OUT_VE.tInAirER_Fan1DemOn.Do AND NOT IN_VE.tERV_OutlAir_Op.Di AND    (IN_VE.bEng_Dem OR IN_VE.tEng_Run.Do), PT:= T#15s);
		xTON_ERV_Outl_Of(IN:= FALSE, PT:= T#5m);
	END_IF;

	bAuxRel_Louvers_OutlAir       := IN_VE.tOutAirER_LouOpened.Di OR Pos_OutlLou1_OK OR Pos_OutlLou2_OK;
	bAuxRel_FireProtFlaps_OutlAir := IN_VE.tFireProtFlap1_OutlAir_Opened.Di AND IN_VE.tFireProtFlap2_OutlAir_Opened.Di;

	xTOF_EngDemEPS(IN:= IN_VE.bEng_Dem_EPS AND NOT IN_VE.tGCB_On.Di, PT:= T#60s);
	bNoMon4BlackStart := xTOF_EngDemEPS.Q AND IN_VE.bEng_Dem_EPS; //T14

	xMsg2296.Enable		:=	IN_VE.tERV_OutlAir_Op.GoodQual;
	xMsg2296.Set		:=	(NOT bNoMon4BlackStart AND ((xTON_ERV_Outl_On.Q AND xTON_StartERV.Q)
							OR  xTON_ERV_Outl_Of.Q))
							OR (IN_VE.bFS_Act AND xTON_StartERV.Q AND NOT bAuxRel_Louvers_OutlAir)
							OR (IN_VE.bFS_Act AND xTON_StartERV.Q AND NOT bAuxRel_FireProtFlaps_OutlAir);
	xMsg2296.PT			:=	T#0s;
	xMsg2296.Prio		:=	3;
	xMsg2296.RiskClass	:=	10;
	xMsg2296.Reset		:=	FALSE;
	xMsg2296();
	MM2VIS.bMsg2296	    :=	xMsg2296.Q;
	(********************************************************************************************************************
	Safety-related application software source code (EN 13849-1 / 4.6.3): END
	*********************************************************************************************************************)

	(*  2630 Air inlet filter difference pressure maximum - engine room ventilation *)
	xMsg2630.Enable	   	:= TRUE;
	xMsg2630.Set       	:= NOT IN_VE.tDPr_InAirFiltERV_Hi.Di;
	xMsg2630.PT		   	:= T#0s;
	xMsg2630.Prio	   	:= 4;
	xMsg2630.RiskClass 	:= 4;
	xMsg2630.Reset	   	:= FALSE;
	xMsg2630();
	MM2VIS.bMsg2630		:= xMsg2630.Q;

	(*  2701 measuring signal failure position air inlet louver 1  *)
	xMsg2701.Enable     := IN_VE.tPB2MM.bSys_Run AND Para.bPos_InlLou1_Active;
	xMsg2701.Set        := IN_VE.tPB2MM.bParaSetupOk AND NOT IN_VE.tPos_InlLou1.GoodQual;
	xMsg2701.PT			:=	T#0s;
	xMsg2701.Prio		:=	4;
	xMsg2701.RiskClass	:=	4;
	xMsg2701.Reset		:=	FALSE;
	xMsg2701();
	MM2VIS.bMsg2701		:=	xMsg2701.Q;
	OUT_VE.bMsg2701		:=	xMsg2701.Q;

	(*  2702 measuring signal failure position air inlet louver 2  *)
	xMsg2702.Enable     := IN_VE.tPB2MM.bSys_Run AND Para.bPos_InlLou2_Active;
	xMsg2702.Set        := IN_VE.tPB2MM.bParaSetupOk AND NOT IN_VE.tPos_InlLou2.GoodQual;
	xMsg2702.PT			:=	T#0s;
	xMsg2702.Prio		:=	4;
	xMsg2702.RiskClass	:=	4;
	xMsg2702.Reset		:=	FALSE;
	xMsg2702();
	MM2VIS.bMsg2702		:=	xMsg2702.Q;
	OUT_VE.bMsg2702		:=	xMsg2702.Q;

	(*  2703 measuring signal failure position air outlet louver 1  *)
	xMsg2703.Enable     := IN_VE.tPB2MM.bSys_Run AND Para.bPos_OutlLou1_Active;
	xMsg2703.Set        := IN_VE.tPB2MM.bParaSetupOk AND NOT IN_VE.tPos_OutlLou1.GoodQual;
	xMsg2703.PT			:=	T#0s;
	xMsg2703.Prio		:=	4;
	xMsg2703.RiskClass	:=	4;
	xMsg2703.Reset		:=	FALSE;
	xMsg2703();
	MM2VIS.bMsg2703		:=	xMsg2703.Q;
	OUT_VE.bMsg2703		:=	xMsg2703.Q;

	(*  2704 measuring signal failure position air outlet louver 2  *)
	xMsg2704.Enable     := IN_VE.tPB2MM.bSys_Run AND Para.bPos_OutlLou2_Active;
	xMsg2704.Set        := IN_VE.tPB2MM.bParaSetupOk AND NOT IN_VE.tPos_OutlLou2.GoodQual;
	xMsg2704.PT			:=	T#0s;
	xMsg2704.Prio		:=	4;
	xMsg2704.RiskClass	:=	4;
	xMsg2704.Reset		:=	FALSE;
	xMsg2704();
	MM2VIS.bMsg2704		:=	xMsg2704.Q;
	OUT_VE.bMsg2704		:=	xMsg2704.Q;

	(*  2705 measuring signal failure engine room difference pressure  *)
	xMsg2705.Enable     := IN_VE.tPB2MM.bSys_Run AND Para.bPrDiff_ER_Active;
	xMsg2705.Set        := IN_VE.tPB2MM.bParaSetupOk AND NOT IN_VE.tPrDiff_ER.GoodQual;
	xMsg2705.PT			:=	T#0s;
	xMsg2705.Prio		:=	4;
	xMsg2705.RiskClass	:=	4;
	xMsg2705.Reset		:=	FALSE;
	xMsg2705();
	MM2VIS.bMsg2705		:=	xMsg2705.Q;
	OUT_VE.bMsg2705		:=	xMsg2705.Q;

	(*  2706 engine room difference pressure low  *)
	xGR_MINR_PrDiff(In := IN_VE.tPrDiff_ER.Ai, Gw:= Para.rPrDiff_ER_Lim_Low, Hy:= Para.rPrDiff_ER_Lim_Low_Hy);
	bPrDiff_Lo := xGR_MINR_PrDiff.Q;

	xMsg2706.Enable     := IN_VE.tPB2MM.bSys_Run AND Para.bPrDiff_ER_Active;
	xMsg2706.Set        := IN_VE.tPB2MM.bParaSetupOk AND bPrDiff_Lo AND IN_VE.tEng_Run.Do;
	xMsg2706.PT			:=	T#10s;
	xMsg2706.Prio		:=	4;
	xMsg2706.RiskClass	:=	4;
	xMsg2706.Reset		:=	FALSE;
	xMsg2706();
	MM2VIS.bMsg2706		:=	xMsg2706.Q;
	OUT_VE.bMsg2706		:=	xMsg2706.Q;

	(*  2707 engine room difference pressure high  *)
	xGR_MAXR_PrDiff(In := IN_VE.tPrDiff_ER.Ai, Gw:= Para.rPrDiff_ER_Lim_High, Hy:= Para.rPrDiff_ER_Lim_High_Hy);
	bPrDiff_Hi := xGR_MAXR_PrDiff.Q;

	xMsg2707.Enable     := IN_VE.tPB2MM.bSys_Run AND Para.bPrDiff_ER_Active;
	xMsg2707.Set        := IN_VE.tPB2MM.bParaSetupOk AND bPrDiff_Hi;
	xMsg2707.PT			:=	T#10s;
	xMsg2707.Prio		:=	4;
	xMsg2707.RiskClass	:=	4;
	xMsg2707.Reset		:=	FALSE;
	xMsg2707();
	MM2VIS.bMsg2707		:=	xMsg2707.Q;
	OUT_VE.bMsg2707		:=	xMsg2707.Q;

	(*  2708 measuring signal failure position air circulation louver 1  *)
	xMsg2708.Enable     := IN_VE.tPB2MM.bSys_Run AND Para.bPos_CircLou1_Active;
	xMsg2708.Set        := IN_VE.tPB2MM.bParaSetupOk AND NOT IN_VE.tPos_CircLou1.GoodQual;
	xMsg2708.PT			:=	T#0s;
	xMsg2708.Prio		:=	4;
	xMsg2708.RiskClass	:=	4;
	xMsg2708.Reset		:=	FALSE;
	xMsg2708();
	MM2VIS.bMsg2708		:=	xMsg2708.Q;
	OUT_VE.bMsg2708		:=	xMsg2708.Q;

	(*  2709 measuring signal failure position air circulation louver 2  *)
	xMsg2709.Enable     := IN_VE.tPB2MM.bSys_Run AND Para.bPos_CircLou2_Active;
	xMsg2709.Set        := IN_VE.tPB2MM.bParaSetupOk AND NOT IN_VE.tPos_CircLou2.GoodQual;
	xMsg2709.PT			:=	T#0s;
	xMsg2709.Prio		:=	4;
	xMsg2709.RiskClass	:=	4;
	xMsg2709.Reset		:=	FALSE;
	xMsg2709();
	MM2VIS.bMsg2709		:=	xMsg2709.Q;
	OUT_VE.bMsg2709		:=	xMsg2709.Q;

	(********************************************************************************************************************
	Safety-related application software source code (EN 13849-1 / 4.6.3): BEGIN
	*********************************************************************************************************************)
	(*  2795 engine room ventilation failure inlet air *)
	IF Para.bInAirER_Fan_FU THEN
		xTON_ERV_In.IN	:= (NOT IN_VE.tER_InlAir_Ext_Err.Di AND IN_VE.tAuxV_Supply_Ok.Di AND IN_VE.tAuxV_Aux_ok.Di)
						OR (    xTON_MonAuxV.Q AND NOT IN_VE.tAuxV_Supply_Ok.Di)
						OR (    xTON_MonAuxV.Q AND NOT IN_VE.tAuxV_Aux_ok.Di);
	ELSE
		xTON_ERV_In.IN	:=  NOT IN_VE.tER_InlAir_Ext_Err.Di;
	END_IF;
	xTON_ERV_In(PT:= T#12s);

	xMsg2795.Enable		:=	TRUE;
	xMsg2795.Set		:=	xTON_ERV_In.Q;
	xMsg2795.PT			:=	T#0s;
	xMsg2795.Prio		:=	4;
	xMsg2795.RiskClass	:=	4;
	xMsg2795.Reset		:=	FALSE;
	xMsg2795();
	MM2VIS.bMsg2795     :=	xMsg2795.Q;
	OUT_VE.bMsg2795     :=  xMsg2795.Q;
	(********************************************************************************************************************
	Safety-related application software source code (EN 13849-1 / 4.6.3): END
	*********************************************************************************************************************)

	(********************************************************************************************************************
	Safety-related application software source code (EN 13849-1 / 4.6.3): BEGIN
	*********************************************************************************************************************)
	(*  2796 engine room ventilation failure outlet air *)
	IF Para.bOutAirER_Fan_FU THEN
		xTON_ERV_Out.IN	:= (NOT IN_VE.tER_OutlAir_Ext_Err.Di AND IN_VE.tAuxV_Supply_Ok.Di AND IN_VE.tAuxV_Aux_ok.Di)
						OR (    xTON_MonAuxV.Q AND NOT IN_VE.tAuxV_Supply_Ok.Di)
						OR (    xTON_MonAuxV.Q AND NOT IN_VE.tAuxV_Aux_ok.Di);
	ELSE
		xTON_ERV_Out.IN	:=  NOT IN_VE.tER_OutlAir_Ext_Err.Di;
	END_IF;
	xTON_ERV_Out(PT:= T#12s);

	xMsg2796.Enable		:=	TRUE;
	xMsg2796.Set		:=	xTON_ERV_Out.Q;
	xMsg2796.PT			:=	T#0s;
	xMsg2796.Prio		:=	4;
	xMsg2796.RiskClass	:=	4;
	xMsg2796.Reset		:=	FALSE;
	xMsg2796();
	MM2VIS.bMsg2796     :=	xMsg2796.Q;
	OUT_VE.bMsg2796     :=  xMsg2796.Q;
	(********************************************************************************************************************
	Safety-related application software source code (EN 13849-1 / 4.6.3): END
	*********************************************************************************************************************)

	(*  2797 parameterization error air inlet louvers *)
	xMsg2797.Enable		:=	TRUE;
	xMsg2797.Set 		:=  NOT (iValueInlLou = 0
							  OR iValueInlLou = 11
							  OR iValueInlLou = 12
							  OR iValueInlLou = 21
	                          OR iValueInlLou = 22);
	xMsg2797.PT			:=	T#2s;
	xMsg2797.Prio		:=	4;
	xMsg2797.RiskClass	:=	4;
	xMsg2797.Reset		:=	FALSE;
	xMsg2797();
	MM2VIS.bMsg2797     :=	xMsg2797.Q;
	OUT_VE.bMsg2797     :=  xMsg2797.Q;

	(*  2798 parameterization error air outlet louvers *)
	xMsg2798.Enable		:=	TRUE;
	xMsg2798.Set 		:=  NOT (iValueOutlLou = 0
							  OR iValueOutlLou = 11
						      OR iValueOutlLou = 12
	                          OR iValueOutlLou = 21
	                          OR iValueOutlLou = 22);
	xMsg2798.PT			:=	T#2s;
	xMsg2798.Prio		:=	4;
	xMsg2798.RiskClass	:=	4;
	xMsg2798.Reset		:=	FALSE;
	xMsg2798();
	MM2VIS.bMsg2798     :=	xMsg2798.Q;
	OUT_VE.bMsg2798     :=  xMsg2798.Q;

	(*  3152 engine room air temperature signal failure *)
	xMsg3152.Enable		:=	IN_VE.tPB2MM.bParaSetupOk AND Para.bT_AirER_Active;
	xMsg3152.Set		:= (NOT IN_VE.tT_AirER.GoodQual AND IN_VE.rT_AirER_Customized <= 0.0)
						OR (	xMsg3152.Q AND IN_VE.bMsg3003 AND bOMSS_MAT);
	xMsg3152.PT			:=	T#0s;
	xMsg3152.Prio		:=	4;
	xMsg3152.RiskClass	:=	4;
	xMsg3152.Reset		:=	FALSE;
	xMsg3152();
	MM2VIS.bMsg3152		:=	xMsg3152.Q;
	OUT_VE.bMsg3152		:=	xMsg3152.Q;

	(*  3223 engine room air inlet temperature signal failure *)						(* --> NOT USED *)
	xMsg3223.Enable		:=	FALSE;
	xMsg3223.Set		:=	FALSE;
	xMsg3223.PT			:=	T#0s;
	xMsg3223.Prio		:=	4;
	xMsg3223.RiskClass	:=	4;
	xMsg3223.Reset		:=	FALSE;
	xMsg3223();
	MM2VIS.bMsg3223		:=	xMsg3223.Q;

	(*  3224 engine room air inlet temperature high *)									(* --> NOT USED *)
	xMsg3224.Enable		:=	FALSE;
	xMsg3224.Set		:=	FALSE;
	xMsg3224.PT			:=	T#0s;
	xMsg3224.Prio		:=	4;
	xMsg3224.RiskClass	:=	4;
	xMsg3224.Reset		:=	FALSE;
	xMsg3224();
	MM2VIS.bMsg3224	    :=	xMsg3224.Q;

	(*---------------------------------------------------------------------------*)
	(*  3302 purge cycle incomplete *)
	xTON_purge(IN:= dmnd_purge AND NOT OUT_VE.bPurgeER_Rdy, PT:= Para.tiPurgeTimeMax);

	xMsg3302.Enable		:=	Para.bPurgecycle_Active;
	xMsg3302.Set		:=	xTON_purge.Q
						OR (dmnd_purge AND IN_VE.tEng_Run.Do AND NOT OUT_VE.bPurgeER_Rdy);
	xMsg3302.PT			:=	T#0s;
	xMsg3302.Prio		:=	2;
	xMsg3302.RiskClass	:=	4;
	xMsg3302.Reset		:=	FALSE;
	xMsg3302();
	MM2VIS.bMsg3302		:=	xMsg3302.Q;

	(********************************************************************************************************************
	Safety-related application software source code (EN 13849-1 / 4.6.3): BEGIN
	*********************************************************************************************************************)
	(*  3367 engine room ventilation failure - doors *)
	xMsg3367.Enable		:=	TRUE;
	xMsg3367.Set		:=	(IN_VE.bEng_Dem OR IN_VE.tEng_Run.Do) AND NOT IN_VE.tER_DoorClosed.Di;
	xMsg3367.PT			:=	T#15s;
	xMsg3367.Prio		:=	3;
	xMsg3367.RiskClass	:=	4;
	xMsg3367.Reset		:=	FALSE;
	xMsg3367();
	MM2VIS.bMsg3367		:=	xMsg3367.Q;
	(********************************************************************************************************************
	Safety-related application software source code (EN 13849-1 / 4.6.3): END
	*********************************************************************************************************************)

	(*---------------------------------------------------------------------------*)
	(*  3571 no release start module from purge cycle *)
	xTON_PurgeNoRel(IN:= IN_VE.bEng_Dem AND NOT IN_VE.tRel_ER_PurgeCycle.Di AND OUT_VE.bPurgeER_Rdy, PT:= T#200s);

	xMsg3571.Enable		:=	Para.bPurgecycle_Active;
	xMsg3571.Set		:=	xTON_PurgeNoRel.Q AND NOT IN_VE.tEng_Run.Do;
	xMsg3571.PT			:=	T#0s;
	xMsg3571.Prio		:=	4;
	xMsg3571.RiskClass	:=	4;
	xMsg3571.Reset		:=	FALSE;
	xMsg3571();
	MM2VIS.bMsg3571		:=	xMsg3571.Q;

	(*---------------------------------------------------------------------------*)
	IF NOT IN_VE.tOutAirER_LouClosed.GoodQual THEN
		IN_VE.tOutAirER_LouClosed.Di  := 	NOT IN_VE.tOutAirER_LouOpened.Di;
	END_IF;
	IF NOT IN_VE.tInAirER_Lou1Closed.GoodQual THEN
		IN_VE.tInAirER_Lou1Closed.Di  :=	NOT IN_VE.tInAirER_Lou1Opened.Di;
	END_IF;
	IF NOT IN_VE.tInAirER_Lou2Closed.GoodQual THEN
		IN_VE.tInAirER_Lou2Closed.Di  :=	NOT IN_VE.tInAirER_Lou2Opened.Di;
	END_IF;

	(* B2968 Air inlet louver position feedback not plausible *)
	TON_InlLou_ssf(IN := IN_VE.tEng_Run.Do AND (
			(IN_VE.tInAirER_Lou1Closed.Di AND IN_VE.tInAirER_Lou1Opened.Di)
		 OR (NOT IN_VE.tInAirER_Lou1Closed.Di AND NOT IN_VE.tInAirER_Lou1Opened.Di)
		 OR (IN_VE.tInAirER_Lou2Closed.Di AND IN_VE.tInAirER_Lou2Opened.Di)
		 OR (NOT IN_VE.tInAirER_Lou2Closed.Di AND NOT IN_VE.tInAirER_Lou2Opened.Di)) , PT := T#2m);

	xMsg2968.Enable	:= TRUE;
	xMsg2968.Set 	:=	NOT Para.bPos_InlLou1_Active AND NOT Para.bPos_InlLou2_Active AND TON_InlLou_ssf.Q;
	xMsg2968.Reset 	:= TRUE;
	xMsg2968();
	MM2VIS.bMsg2968   := xMsg2968.Q;

	(* B2969 Air outlet louver position feedback not plausible *)
	TON_OutLou_ssf(IN := IN_VE.tEng_Run.Do AND ((IN_VE.tOutAirER_LouClosed.Di AND IN_VE.tOutAirER_LouOpened.Di)
		 OR ((NOT IN_VE.tOutAirER_LouClosed.Di AND NOT IN_VE.tOutAirER_LouOpened.Di))) , PT := T#2m);

	xMsg2969.Enable	:= TRUE;
	xMsg2969.Set 	:=	NOT Para.bPos_OutlLou1_Active AND NOT Para.bPos_OutlLou2_Active AND TON_OutLou_ssf.Q;
	xMsg2969.Reset := TRUE;
	xMsg2969();
	MM2VIS.bMsg2969   := xMsg2969.Q;
	(*---------------------------------------------------------------------------*)
	(*  9401 Louver failure *)

	IF Para.bER_VentColdCountryMode THEN
		bLouvers := IN_VE.tOutAirER_LouOpened.Di;
	ELSE
		IF IN_VE.bFS_Act AND NOT xTON_MonFS.Q THEN
			bLouvers := (IN_VE.tOutAirER_LouOpened.Di OR NOT IN_VE.tOutAirER_LouClosed.Di OR Pos_OutlLou1_OK OR Pos_OutlLou2_OK) AND
									(IN_VE.tInAirER_Lou1Opened.Di OR NOT IN_VE.tInAirER_Lou1Closed.Di OR Pos_InlLou1_OK  OR Pos_InlLou2_OK);
		ELSE
			bLouvers := (IN_VE.tOutAirER_LouOpened.Di OR Pos_OutlLou1_OK OR Pos_OutlLou2_OK) AND
									(IN_VE.tInAirER_Lou1Opened.Di OR Pos_InlLou1_OK  OR Pos_InlLou2_OK);
		END_IF;
	END_IF;

	(*  wait until louvers ready or 160s which is max time for the slowest SF24A-SR-S2 louver*)
	IF bLouvers THEN
		xTON_Wait_louver	(IN	:= IN_VE.bEng_Aux_Dem, PT:=T#0s);
	ELSE
		xTON_Wait_louver	(IN	:= IN_VE.bEng_Aux_Dem, PT:= T#160s);
	END_IF

	xMsg9401.Enable		:=	TRUE;
	xMsg9401.Set		:=	xTON_Wait_louver.Q  AND (NOT bLouvers AND IN_VE.bEng_Aux_Dem);
	xMsg9401.PT			:=	T#0s;
	xMsg9401.Prio		:=	3;
	xMsg9401.RiskClass	:=	4;
	xMsg9401.Reset		:=	FALSE;
	xMsg9401();
	MM2VIS.bMsg9401		:=	xMsg9401.Q;
	(*---------------------------------------------------------------------------*)
	(* operating messages > AMM *)
	// bMsg0000	:=	NOT TRUE;						(* Bxxxx operating message text *)
	// bMsg0001	:=		FALSE;						(* Bxxxx operating message text *)

	(*---------------------------------------------------------------------------*)
	(* general alarms for further module operations *)
	bGnlTrip1	:=	OUT_VE.tVE2AB.bGnlTrip1 	OR IN_VE.tAB2VE.bGnlTrip1;
	bGnlTrip2	:=	OUT_VE.tVE2AB.bGnlTrip2 	OR IN_VE.tAB2VE.bGnlTrip2;
	bGnlTrip3	:=	OUT_VE.tVE2AB.bGnlTrip3 	OR IN_VE.tAB2VE.bGnlTrip3;
	bGnlWarning :=	OUT_VE.tVE2AB.bGnlWarning 	OR IN_VE.tAB2VE.bGnlWarning;

	bGnlTrip	:= bGnlTrip1 OR bGnlTrip2 OR bGnlTrip3;
	(*******************************************************************************)
END_PROGRAM
```

#### MsgVEInit.st
```iecst
(*******************************************************************************
Msg_VE	 			 alarms generation

This code is confidential and proprietary to the INNIO Company.
It may not be used in any form, or reproduced in any manner,
without written permission of the INNIO Company.
Copyright, INNIO Company, 2019

Customized modifications: -
------------------------

History:
-------
V0.00.0	29.07.2011	lettenb.	new
V4.06.0	16.07.2018	Perktold,	2968 and 2969 Air inlet/outlet louver status signal failure added

Instructions for use:
--------------------
1) declare alarm with function block "Msg"

2) use template to create a new alarm, substitue 0000 by message number:

	xMsg0000.Num		:=	0000;					alarm number
	xMsg0000.AmmSysAdr	:=  iAdrAmmBase2MM;			do not change
	xMsg0000.AmmOutAdr	:=  iAdrMM2AmmBase;			do not change

3) 	set alarm number

Outstandings:
------------
(*******************************************************************************)
PROGRAM _INIT

	iAdrAmmBase2MM		:=  ADR(IN_VE.tAB2VE);
	iAdrMM2AmmBase		:=  ADR(OUT_VE.tVE2AB);

	(*---------------------------------------------------------------------------*)
	xMsg1135.Num		:=	1135;
	xMsg1135.AmmInAdr	:=  iAdrAmmBase2MM;
	xMsg1135.AmmOutAdr	:=  iAdrMM2AmmBase;

	xMsg1138.Num		:=	1138;
	xMsg1138.AmmInAdr	:=  iAdrAmmBase2MM;
	xMsg1138.AmmOutAdr	:=  iAdrMM2AmmBase;

	xMsg2120.Num		:=	2120;
	xMsg2120.AmmInAdr	:=  iAdrAmmBase2MM;
	xMsg2120.AmmOutAdr	:=  iAdrMM2AmmBase;

	xMsg2295.Num		:=	2295;
	xMsg2295.AmmInAdr	:=  iAdrAmmBase2MM;
	xMsg2295.AmmOutAdr	:=  iAdrMM2AmmBase;

	xMsg2296.Num		:=	2296;
	xMsg2296.AmmInAdr	:=  iAdrAmmBase2MM;
	xMsg2296.AmmOutAdr	:=  iAdrMM2AmmBase;

	xMsg2472.Num		:=	2472;
	xMsg2472.AmmInAdr	:=  iAdrAmmBase2MM;
	xMsg2472.AmmOutAdr	:=  iAdrMM2AmmBase;

	xMsg2630.Num		:=	2630;
	xMsg2630.AmmInAdr	:=  iAdrAmmBase2MM;
	xMsg2630.AmmOutAdr	:=  iAdrMM2AmmBase;

	xMsg2701.Num		:=	2701;
	xMsg2701.AmmInAdr	:=  iAdrAmmBase2MM;
	xMsg2701.AmmOutAdr	:=  iAdrMM2AmmBase;

	xMsg2702.Num		:=	2702;
	xMsg2702.AmmInAdr	:=  iAdrAmmBase2MM;
	xMsg2702.AmmOutAdr	:=  iAdrMM2AmmBase;

	xMsg2703.Num		:=	2703;
	xMsg2703.AmmInAdr	:=  iAdrAmmBase2MM;
	xMsg2703.AmmOutAdr	:=  iAdrMM2AmmBase;

	xMsg2704.Num		:=	2704;
	xMsg2704.AmmInAdr	:=  iAdrAmmBase2MM;
	xMsg2704.AmmOutAdr	:=  iAdrMM2AmmBase;

	xMsg2705.Num		:=	2705;
	xMsg2705.AmmInAdr	:=  iAdrAmmBase2MM;
	xMsg2705.AmmOutAdr	:=  iAdrMM2AmmBase;

	xMsg2706.Num		:=	2706;
	xMsg2706.AmmInAdr	:=  iAdrAmmBase2MM;
	xMsg2706.AmmOutAdr	:=  iAdrMM2AmmBase;

	xMsg2707.Num		:=	2707;
	xMsg2707.AmmInAdr	:=  iAdrAmmBase2MM;
	xMsg2707.AmmOutAdr	:=  iAdrMM2AmmBase;

	xMsg2708.Num		:=	2708;
	xMsg2708.AmmInAdr	:=  iAdrAmmBase2MM;
	xMsg2708.AmmOutAdr	:=  iAdrMM2AmmBase;

	xMsg2709.Num		:=	2709;
	xMsg2709.AmmInAdr	:=  iAdrAmmBase2MM;
	xMsg2709.AmmOutAdr	:=  iAdrMM2AmmBase;

	xMsg2795.Num		:=	2795;
	xMsg2795.AmmInAdr	:=  iAdrAmmBase2MM;
	xMsg2795.AmmOutAdr	:=  iAdrMM2AmmBase;

	xMsg2796.Num		:=	2796;
	xMsg2796.AmmInAdr	:=  iAdrAmmBase2MM;
	xMsg2796.AmmOutAdr	:=  iAdrMM2AmmBase;

	xMsg2797.Num		:=	2797;
	xMsg2797.AmmInAdr	:=  iAdrAmmBase2MM;
	xMsg2797.AmmOutAdr	:=  iAdrMM2AmmBase;

	xMsg2798.Num		:=	2798;
	xMsg2798.AmmInAdr	:=  iAdrAmmBase2MM;
	xMsg2798.AmmOutAdr	:=  iAdrMM2AmmBase;

	xMsg3152.Num		:=	3152;
	xMsg3152.AmmInAdr	:=  iAdrAmmBase2MM;
	xMsg3152.AmmOutAdr	:=  iAdrMM2AmmBase;

	xMsg3223.Num		:=	3223;
	xMsg3223.AmmInAdr	:=  iAdrAmmBase2MM;
	xMsg3223.AmmOutAdr	:=  iAdrMM2AmmBase;

	xMsg3224.Num		:=	3224;
	xMsg3224.AmmInAdr	:=  iAdrAmmBase2MM;
	xMsg3224.AmmOutAdr	:=  iAdrMM2AmmBase;

	xMsg3302.Num		:=	3302;
	xMsg3302.AmmInAdr	:=  iAdrAmmBase2MM;
	xMsg3302.AmmOutAdr	:=  iAdrMM2AmmBase;

	xMsg3367.Num		:=	3367;
	xMsg3367.AmmInAdr	:=  iAdrAmmBase2MM;
	xMsg3367.AmmOutAdr	:=  iAdrMM2AmmBase;

	xMsg3571.Num		:=	3571;
	xMsg3571.AmmInAdr	:=  iAdrAmmBase2MM;
	xMsg3571.AmmOutAdr	:=  iAdrMM2AmmBase;

	xMsg9401.Num		:=	9401;
	xMsg9401.AmmInAdr	:=  iAdrAmmBase2MM;
	xMsg9401.AmmOutAdr	:=  iAdrMM2AmmBase;

(* B2968 Air inlet louver position feedback not plausible *)
	xMsg2968.Num		:=	2968;
	xMsg2968.AmmInAdr	:=  iAdrAmmBase2MM;
	xMsg2968.AmmOutAdr	:=  iAdrMM2AmmBase;

(* B2969 Air outlet louver position feedback not plausible *)
	xMsg2969.Num		:=	2969;
	xMsg2969.AmmInAdr	:=  iAdrAmmBase2MM;
	xMsg2969.AmmOutAdr	:=  iAdrMM2AmmBase;

//	xMsg0000.Num		:=	0000;
//	xMsg0000.AmmInAdr	:=  iAdrAmmBase2MM;
//	xMsg0000.AmmOutAdr	:=  iAdrMM2AmmBase;

END_PROGRAM
```

#### MsgVE.var
```iecst
VAR
	bAuxRel_Louvers_OutlAir : BOOL; (*Release auxiliaries from outlet air louvers*)
	bAuxRel_FireProtFlaps_OutlAir : BOOL; (*Release auxiliaires from outlet air fire protection flaps*)
	bAuxRel_Louvers_InlAir : BOOL; (*Release auxiliaries from inlet air louvers*)
	bAuxRel_FireProtFlaps_InlAir : BOOL; (*Release auxiliaires from inlet air fire protection flaps*)
	bLouvers : BOOL; (*Louver status*)
	bAuxRel_FireProtFlaps : BOOL; (*Release auxiliaires from  protection flaps*)
	xGR_MINR_PrDiff : GR_MINR := (0); (*Limit low for engine room difference pressure *)
	xGR_MAXR_PrDiff : GR_MAXR := (0); (*Limit high for engine room difference pressure*)
	bPrDiff_Hi : BOOL; (*Limit high reached*)
	bPrDiff_Lo : BOOL; (*Limit low reached*)
	xTON_ERV_On : TON;
	xTON_ERV_Of : TON;
	xTON_ERV_Inl_On : TON;
	xTON_ERV_Inl_Of : TON;
	xTON_ERV_Outl_On : TON;
	xTON_ERV_Outl_Of : TON;
	xTON_MonAuxV : TON;
	xTON_RoomTemp : TON;
	T_RTM : BOOL;
	RTM_VISA : BOOL;
	xTON_purge : TON;
	xTON_PurgeNoRel : TON;
	iAdrAmmBase2MM : UDINT;
	iAdrMM2AmmBase : UDINT;
	xTON_StartERV : TON;
	bERV_AirFlowMon_Off : BOOL; (*ERV air flow monitoring off*)
	bERV_InlAirFlowMon_Off : BOOL; (*ERV inlet air flow monitoring off*)
	bERV_OutlAirFlowMon_Off : BOOL; (*ERV outlet air flow monitoring off*)
	bNoMon4BlackStart : BOOL;
	xTOF_EngDemEPS : TOF;
	bAuxRel_Louvers : BOOL;
	xMsg1135 : Msg;
	xMsg1138 : Msg;
	xMsg2120 : Msg;
	xMsg2295 : Msg;
	xMsg2296 : Msg;
	xMsg2630 : Msg;
	xMsg2701 : Msg;
	xMsg2702 : Msg;
	xMsg2703 : Msg;
	xMsg2704 : Msg;
	xMsg2705 : Msg;
	xMsg2706 : Msg;
	xMsg2707 : Msg;
	xMsg2708 : Msg;
	xMsg2709 : Msg;
	xMsg2795 : Msg;
	xMsg2796 : Msg;
	xMsg2797 : Msg;
	xMsg2798 : Msg;
	xMsg3152 : Msg;
	xMsg3223 : Msg;
	xMsg3224 : Msg;
	xMsg3302 : Msg;
	xMsg3367 : Msg;
	xMsg3571 : Msg;
	TON_InlLou_ssf : TON;
	TON_OutLou_ssf : TON;
	xTON_ERV : TON;
	xTON_ERV_In : TON;
	xTON_ERV_Out : TON;
	xMsg2968 : Msg; (* B2968 Air inlet louver position feedback not plausible *)
	xMsg2969 : Msg; (* B2969 Air outlet louver position feedback not plausible *)
	xMsg2472 : Msg; (* B2472 Engine room temperature high warning*)
	xMsg9401 : Msg; (* A9401 Louvers failure*)
	xTON_InAirER_LouFail : TON; (* Inlet louver required and not opened*)
	xTON_MonFS : TON;
	xTON_Wait_louver : TON;  (*Wait for louver*)
END_VAR
```

### Program Logical/Ventilation/ParVE (IEC, version 4.06.0) - + parameter handling

- perm_par.st (not readable text: treated as protected, skipped)

#### perm_par.var
```iecst
VAR
	tParaIntern : ParaHandler_typ; (*Connector type to perm_par*)
	tMM2ParaBase_ReadBack : MM2ParaBase_type; (*INTERNAL! V4.06 new readback structure for information from previous tasks*)
	bWriteDataObj : BOOL; (* TRUE=write data object module *)
	bDataObjLenErr : BOOL; (*Error occured in permem: data module size missmatch*)
	bCreateDataObj : BOOL; (* TRUE=create new data object *)
	bWriteOnce : BOOL; (* write permanent memory once *)
	DatObjCreate_01 : DatObjCreate; (* data object create *)
	DatObjInfoBak_02 : DatObjInfo; (* data object info *)
	DatObjDelete_01 : DatObjDelete; (* data object delete *)
	DatObjRead_01 : DatObjRead; (* data object read *)
	DatObjRead_02 : DatObjRead; (* manual initiated data object read *)
	DatObjWrite_01 : DatObjWrite; (* data object write *)
	DatObjDelete_02 : DatObjDelete; (* data object delete *)
	DatObjDelete_11 : DatObjDelete; (*Delete Backup File*)
	DatObjInfo_01 : DatObjInfo; (* data object info *)
	DatObjInfo_02 : DatObjInfo; (* data object info *)
	szModuleName : STRING[35]; (* module name of object *)
	szModuleNameBackup : STRING[35]; (* module name of posiibly created backup object *)
	DatObjCopy_01 : DatObjCopy;
	bCopyDataObj : BOOL;
	TON_WarnDelay : TON;
	TON_WritePMEM : TON; (* delay write permanent memory *)
	ulPMPointer : UDINT; (* adress of actual checksum value *)
	ulChecksum : UDINT; (* parameter checksum value *)
	pm_len : UDINT; (* permanent value lenght *)
	ulChecksumOld : UDINT; (* last vlaue of parameter checksum *)
	ulChkValue : UDINT; (* actual value of parameter pointer *)
	pm_id : UDINT; (* permanent value identifier *)
	pm_p : UDINT; (* permanent value pointer *)
	DatObjInfo_META : DatObjInfo;
	DatObjRead_META : DatObjRead;
	szMetaDataRaw : STRING[2000];
	szMetaData : ARRAY[0..4] OF STRING[35];
	szMetaDataVis : ARRAY[0..3] OF STRING[35];
	ssIndex : INT;
	ssCount : INT;
	ucMetaDataRaw : ARRAY[0..2000] OF USINT;
	ssCount2 : INT;
	szMetaDataFile : STRING[10];
	szText1 : STRING[20];
	pv_adr_IN_XX_tPB2MM : UDINT;
	pv_lng : UDINT;
	pv_lng_IN_XX_tPB2MM : UDINT;
	pv_lng_OUT_XX_tPB2MM : UDINT;
	szText2 : STRING[20];
	pv_adr_OUT_XX_tXX2PB : UDINT;
END_VAR
VAR CONSTANT
	ERR_NOERROR : UINT := 0;
END_VAR
VAR
	usPMWriteCnt : UINT;
	pm_Error : UDINT; (* permanent value error *) (* Deleted: pm : ParaMem_typ; permanent memory tags mathias, 22.8.11*)
	fun_Error : UDINT := 0; (*state > 0 = function error*)
	xLocalParaCheck : ParaCheckFUB; (*local function instance to check parameter values*)
	TON_ParaSetupOk : TON;
	bParaCheckSystemOk : BOOL;
	iDebug_ParaOkChecked : UDINT;
	bRestoreBackupDataObj : BOOL := FALSE;
	bRestoreDataObjContent : BOOL := FALSE;
	pm_id_backup : UDINT;
	pm_p_Backup : UDINT;
	DatObjCopy_02 : DatObjCopy;
	bDeleteBackupDataObj : BOOL := FALSE; (*Command to delete backup data module file on purpose*)
	bDebugPara : ARRAY[0..5] OF BOOL;
	ssIndex2 : INT;
	ssIndex3 : INT;
	ssIndex4 : INT;
	ssIndexVis : INT;
	szText : STRING[40];
	pv_adr_Para : UDINT;
	szParaSnippet : ARRAY[0..5] OF STRING[150];
	szParaIndex : STRING[10];
	slValue : DINT;
	iModuleDLD_ResetCount : INT;
	bDownloadDetected : BOOL;
	bFlagParaStructCopyWorking : BOOL; (*true, if cyclic para copying is active, 1 false cycle at every copy *)
	bStoreInitParaInDataObj : BOOL := FALSE;
	bTestflag : BOOL;
	bReadOutMETA_Once : BOOL;
	tParaCheck_iPvAdress : ARRAY[0..5] OF UDINT;
	tParaCheck_iPvLengt : ARRAY[0..5] OF UDINT;
	tParaCheck_rPvValue : ARRAY[0..5] OF REAL;
	tParaCheck_rRangeMIN : ARRAY[0..5] OF REAL;
	tParaCheck_rRangeMAX : ARRAY[0..5] OF REAL;
	tParaCheck_szPvName : ARRAY[0..5] OF STRING[35];
	ssFormatDetected : INT;
	szMetaDataPart : STRING[150];
	szFullTaskName : STRING[35];
	szFullMetaModuleName : STRING[35];
	debugLen : INT;
	debugSize : INT := 0;
	strcat_adr1 : UDINT;
	strcat_adr2 : UDINT;
	ssIndexTN : INT;
	bAlternate : BOOL;
	n : INT;
	iAlternateChecksum : DINT;
	iAlternateChecksumOld : DINT;
	ulDebugChkValue : ARRAY[0..999] OF UDINT;
	Adr1 : UDINT;
	Adr2 : UDINT;
	usPMWriteCntStepsize : UINT := 1; (*different step sizes to help debug*)
	usPMWriteCntXOR : UINT;
	usPMWriteCntAltSum : UINT;
	ulAdrPM : UDINT;
	usChkValuePM : USINT;
	ulAdrPara : UDINT;
	ulPara_len : UDINT;
	usChkValuePara : USINT;
	iDebugCountPMDifferences : DINT := 0;
	bEngineRunDetected : BOOL; (*detection status bit autocommand 100 /101  for engine run state*)
	ucMetaDataDebugInfoLine : ARRAY[0..24] OF STRING[80];
	ssIndexMand : INT := 0;
	szMetaDataMand : STRING[35];
	iMyErrorInfo_Autoreset : DINT; (*internal autoreset counter*)
	ssIndex_Version : INT; (*internal*)
	ssIndex_BU : INT; (*internal*)
	ssIndex_BU2 : INT; (*internal*)
END_VAR
```

- Visualisation Logical/Visu (not shown)

### Package Logical/CBM - CB: CBM

### Data object Logical/CBM/META_CB (Simple) - MODUL META data file

#### META_CB.dat
```
; *******************************************************************************
; AGGR: Module Meta Data (data module)
;
; This code is confidential and proprietary to the INNIO Company.
; It may not be used in any form, or reproduced in any manner, without the express
; written permission of the INNIO Company.
; Copyright, INNIO Company, 2025
;
; Customized modifications: -
; ------------------------
;
; History:
; -------
; V03.99.00.00	06.03.2013	Weitzer		generated for modular software
; V03.99.02.00	29.05.2013	Zengerer	initial dependencies prepared
; V04.00.00.00	30.01.2014	Denk		new version
; V04.02.00.00	20.02.2015	Caks,		introduction of CBM module
; V04.03.00.00	10.11.2015	Caks,		added mandatory statement
;				13.11.2015	Waldhart,	added place holder tasks
; V04.04.00.00	20.03.2017	Waldhart,	ATD package implemented
; V04.05.00.00	27.11.2017	Waldhart,	newest Version from IMEP based friciton monitoring V0.4.3
;				14.02.2017	Waldhart,	PBCMem new implemented
;				26.02.2018	502423184	Statistic package update
; V04.06.00.00	16.03.2018	502423184,	new ECB, TCB, ErrCnt & Statistic file generation
; V04.06.01.00	16.11.2018	502423184,	release version, removed clock_ms()
; V04.07.00.00	22.03.2019	Waldhart,	IMEP based friciton monitoring V0.06.0
;										ECB, TCB content increased
; V04.09.00.00	30.08.2019	Waldhart,	Permanent dataobject added
;				23.01.2020	Schmidt,	GEN2diag: added interface for deactivation when LX2 is switched off
;				17.04.2020	Waldhart,	declared but unused PV`s deleted
; V04.10.00.00	22.07.2020	Schmidt,	IMEP based friciton monitoring V0.07.1
; V04.11.00.00	08.11.2021	Keller, 	Gen2 gas quality offset
;				01.12.2021	Kafka,		Lambda Controller PBC, increase buffer size
; V04.12.00.00	10.05.2022	Schmidt, 	GEN2diag: increased delay for first activation to avoid FP detections while in GEN2 lambda minimum (issue #806)
;				08.09.2022	Andre,		Select the engine speed from the ICxx module also if SEMIC is active
; 				16.01.2023	Kafka,		Correct conversion factors for ECBMem and TCBMem dataitems
; V04.13.00.00	19.10.2023	Schmidt, 	GEN2diag: for PBC deactivate monitoring during misfire (issue #1076)
;               30.10.2023	Kafka,		CBM HMI Handshake added, solve special sign issue
;               24.11.2023  Bachler,    Add bGridStat_GridLoss trigger
;				07.12.2023	Schmidt,	Added combustion anomaly detection information to statistic
; V04.14.00.00	22.07.2024	Kafka,		Remove G2 signals, increase buffer for KLS and PBC data
;				19.10.2024	Vigh, 		Added exhaust fast pressure value to TCB_MEM
;				14.03.2025	Perktold	Clean up, added Ti_Purge_Dur and Ti_Wait4StartTempRel to start statistic
;
; Instructions for use:
; --------------------
; make only changes at the version numbers
;
; Outstandings:
; ------------
;
; *******************************************************************************
;
"<META>"
;
; Module ID: 25187
"<MODUL>CB</MODUL>"
;
; Module Version (xx.yy.zz.cc)
"<VERSION>04.14.00.00</VERSION>"
;
; Module Basisupdate Version BU (00-99)
"<BASISUPDATE_VERSION>00</BASISUPDATE_VERSION>"
;
; Optional: specify order number for limitated module usage
"<ORDER></ORDER>" ;<!--(optional for restricted customizations; missing statement makes module valid for all orders)-->
;
; Parameter Check <PARAn Name='aAbcdef' MIN='xxx' MAX='yyy' />  (watch for correct spacings and apostrophs!)
"<PARAMETER_CHK>"
"<PARA1 Name='iEng_Motortype' MIN='208' MAX='920' />"
"<PARA2 />"
"<PARA3 />"
"<PARA4 />"
"<PARA5 />"
"</PARAMETER_CHK>"
;
; Statement, if engine operation is also allowed without this module (FALSE) or if this module´s parameter check passing is mandatory (TRUE)
"<MANDATORYMODULE>TRUE</MANDATORYMODULE>"
;
; Permanent Datamodule Filenames<!-- NAME ist ohne Dateiendung einzutragen; Nur für Counter und interne Parameter verwenden-->
"<DATAMODULES>" ;<!-- optional; mehrere DATAMODULES erlaubt-->
"	<DATAMODULE>par_CB</DATAMODULE>"
"	<DATAMODULE>Stats_perm</DATAMODULE>"
"	<DATAMODULE>FDT_perm</DATAMODULE>"
"	<DATAMODULE>LOM_perm</DATAMODULE>"
"	<DATAMODULE>FAM_perm</DATAMODULE>"
"	<DATAMODULE>FAMST_perm</DATAMODULE>"
"	<DATAMODULE>CBM_perm</DATAMODULE>"
"</DATAMODULES>"
;
; Dependencies Modules (MMxx.yy.zz.cc)
"<DEPENDENCIES>"
"	<DEPENDENCY MODULE='HA' VERSION='04.07.00.00' />"
"	<DEPENDENCY MODULE='SA' VERSION='04.11.00.00' />"
"	<DEPENDENCY MODULE='EC' VERSION='04.14.00.00' />"
"	<DEPENDENCY MODULE='PB' VERSION='04.06.00.00' />"	;new permanent file info
"	<DEPENDENCY MODULE='AB' VERSION='04.07.00.00' />"    ; for iMsg array V4.07
"	<DEPENDENCY MODULE='CU' VERSION='04.00.00.00' />"    ; corrected for SW download via HMI
"	<DEPENDENCY MODULE='GT' VERSION='04.00.00.00' />"    ; corrected for SW download via HMI
"	<DEPENDENCY MODULE='GD' VERSION='04.00.00.00' />"    ; corrected for SW download via HMI
"	<DEPENDENCY MODULE='EG' VERSION='04.00.00.00' />"    ; corrected for SW download via HMI
"	<DEPENDENCY MODULE='OP' VERSION='04.00.00.00' />"    ; corrected for SW download via HMI
"	<DEPENDENCY MODULE='CH' VERSION='04.00.00.00' />"    ; corrected for SW download via HMI
"	<DEPENDENCY MODULE='IC' VERSION='04.00.00.00' />"    ; corrected for SW download via HMI
"	<DEPENDENCY MODULE='EM' VERSION='04.00.00.00' />"    ; corrected for SW download via HMI
"	<DEPENDENCY MODULE='IG' VERSION='04.00.00.00' />"    ; corrected for SW download via HMI
"	<DEPENDENCY MODULE='SY' VERSION='04.00.00.00' />"    ; corrected for SW download via HMI
"	<DEPENDENCY MODULE='AG' VERSION='04.14.00.00' />"    ; corrected for SW download via HMI
"	<DEPENDENCY MODULE='KN' VERSION='04.00.00.00' />"    ; corrected for SW download via HMI
"	<DEPENDENCY MODULE='EX' VERSION='04.00.00.00' />"    ; corrected for SW download via HMI
"	<DEPENDENCY MODULE='VI' VERSION='04.00.00.00' />"    ; corrected for SW download via HMI
"   <DEPENDENCY VISVERSION='02.15.00.00' />"			; Dependencies Visualization
"</DEPENDENCIES>"
;
; Module function description
"<MODULEFUNCTION>" ;<!-- short overview documentation of module function; add reference to detailed information, if available-->
"	<General>	"
"	Please ask the module owner to enter a general module description here. "
"	</General>	"
""
"	<F1 Name='enter name of main function 1 here' LastModified='04.00.00.00'>"
"	Enter function 1 description for module here.	"
"	</F1>"
"	<F3 Name='enter name of main function 2 here' LastModified='04.00.00.00'>"
"	Enter function 2 description for module here.	"
"	</F2>"
"	<F3 Name='enter name of main function 3 here' LastModified='04.00.00.00'>"
"	Enter function 3 description for module here.	"
"	</F3>"
""
"	<Info>"
"	Please enter additional module info here.	"
"	</Info>"
""
"	<Customized LastModified='4.0.0.0'>	"
"	- Nothing "
"	</Customized>	"
""
"</MODULEFUNCTION>"
;
"</META>"
```
